(* Logix 5000 project; controller NSH_PLC1 vendor 1 type 14 code 167 rev 32.11; software revision 32.02; part 9 of 12 *)
(* tags used below, declared in another part *)
   DummyOutput : BOOL;
   LS101 : BOOL;   // Dummy Limit Switch
   MainBin1 : MainBins;   // PreClean to Huller, Main Bin #1
   MainBin2 : MainBins;   // PreClean to Huller, Main Bin #1
   MainBin3 : MainBins;   // PreClean to Huller, Main Bin #1
   MainBin4 : MainBins;   // PreClean to Huller, Main Bin #1
   MainBin5 : MainBins;   // PreClean to Huller, Main Bin #1
   MainBin6 : MainBins;   // PreClean to Huller, Main Bin #1
   MainBin7 : MainBins;   // PreClean to Huller, Main Bin #1
   MainBin8 : MainBins;   // PreClean to Huller, Main Bin #1
(* MainProgram, continued *)

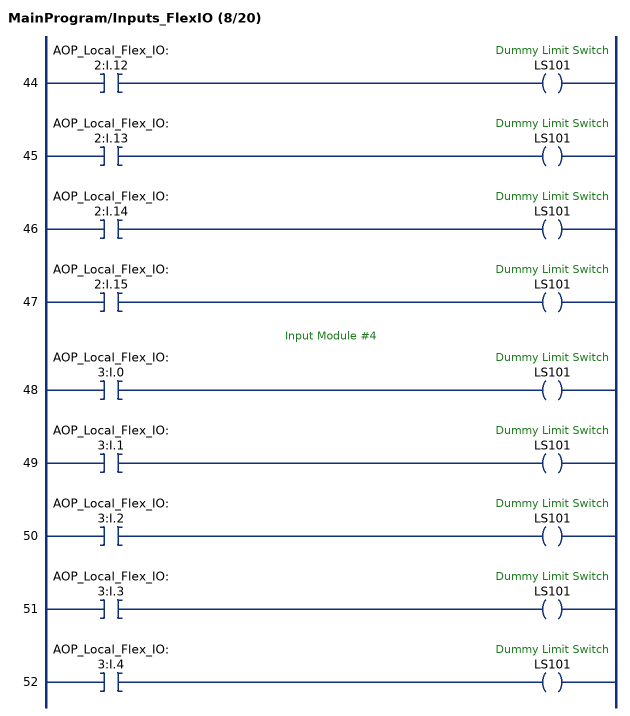
   44: XIC(AOP_Local_Flex_IO:2:I.12)OTE(LS101);
   45: XIC(AOP_Local_Flex_IO:2:I.13)OTE(LS101);
   46: XIC(AOP_Local_Flex_IO:2:I.14)OTE(LS101);
   47: XIC(AOP_Local_Flex_IO:2:I.15)OTE(LS101);
   // Input Module #4
   48: XIC(AOP_Local_Flex_IO:3:I.0)OTE(LS101);
   49: XIC(AOP_Local_Flex_IO:3:I.1)OTE(LS101);
   50: XIC(AOP_Local_Flex_IO:3:I.2)OTE(LS101);
   51: XIC(AOP_Local_Flex_IO:3:I.3)OTE(LS101);
   52: XIC(AOP_Local_Flex_IO:3:I.4)OTE(LS101);
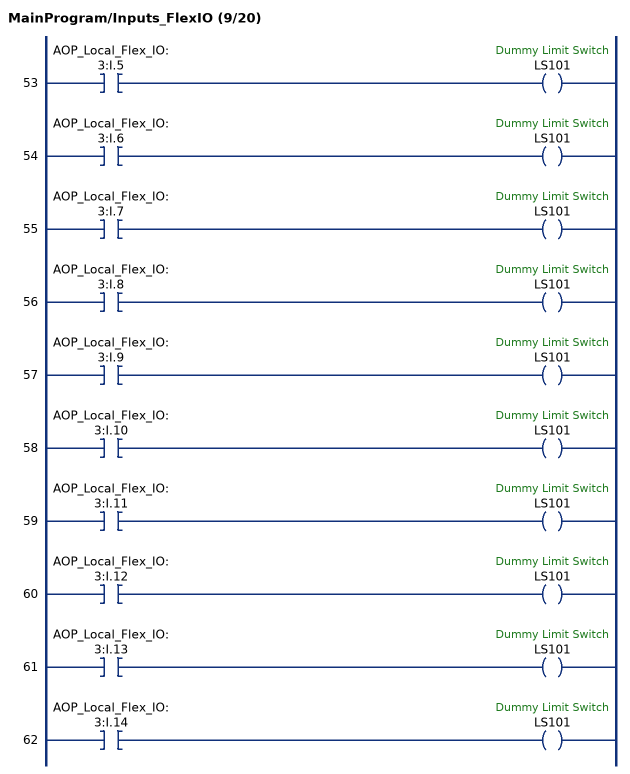
   53: XIC(AOP_Local_Flex_IO:3:I.5)OTE(LS101);
   54: XIC(AOP_Local_Flex_IO:3:I.6)OTE(LS101);
   55: XIC(AOP_Local_Flex_IO:3:I.7)OTE(LS101);
   56: XIC(AOP_Local_Flex_IO:3:I.8)OTE(LS101);
   57: XIC(AOP_Local_Flex_IO:3:I.9)OTE(LS101);
   58: XIC(AOP_Local_Flex_IO:3:I.10)OTE(LS101);
   59: XIC(AOP_Local_Flex_IO:3:I.11)OTE(LS101);
   60: XIC(AOP_Local_Flex_IO:3:I.12)OTE(LS101);
   61: XIC(AOP_Local_Flex_IO:3:I.13)OTE(LS101);
   62: XIC(AOP_Local_Flex_IO:3:I.14)OTE(LS101);
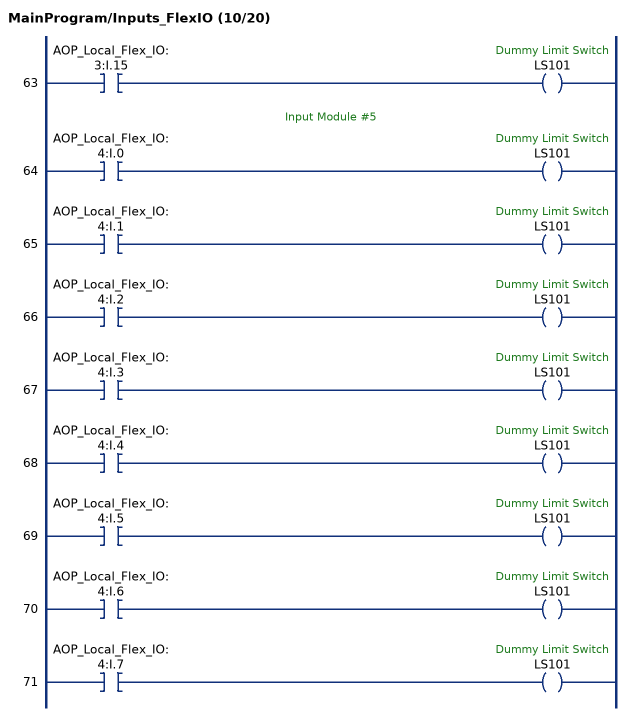
   63: XIC(AOP_Local_Flex_IO:3:I.15)OTE(LS101);
   // Input Module #5
   64: XIC(AOP_Local_Flex_IO:4:I.0)OTE(LS101);
   65: XIC(AOP_Local_Flex_IO:4:I.1)OTE(LS101);
   66: XIC(AOP_Local_Flex_IO:4:I.2)OTE(LS101);
   67: XIC(AOP_Local_Flex_IO:4:I.3)OTE(LS101);
   68: XIC(AOP_Local_Flex_IO:4:I.4)OTE(LS101);
   69: XIC(AOP_Local_Flex_IO:4:I.5)OTE(LS101);
   70: XIC(AOP_Local_Flex_IO:4:I.6)OTE(LS101);
   71: XIC(AOP_Local_Flex_IO:4:I.7)OTE(LS101);
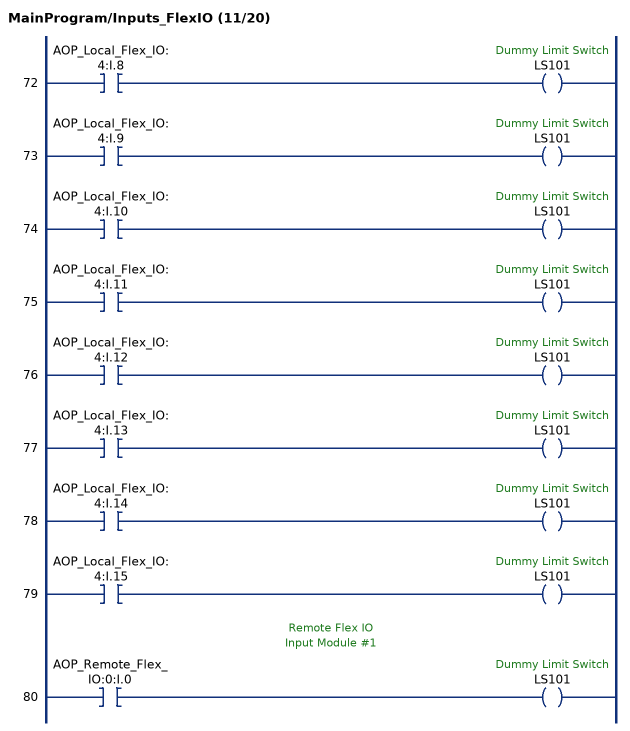
   72: XIC(AOP_Local_Flex_IO:4:I.8)OTE(LS101);
   73: XIC(AOP_Local_Flex_IO:4:I.9)OTE(LS101);
   74: XIC(AOP_Local_Flex_IO:4:I.10)OTE(LS101);
   75: XIC(AOP_Local_Flex_IO:4:I.11)OTE(LS101);
   76: XIC(AOP_Local_Flex_IO:4:I.12)OTE(LS101);
   77: XIC(AOP_Local_Flex_IO:4:I.13)OTE(LS101);
   78: XIC(AOP_Local_Flex_IO:4:I.14)OTE(LS101);
   79: XIC(AOP_Local_Flex_IO:4:I.15)OTE(LS101);
   // Remote Flex IO
   // Input Module #1
   80: XIC(AOP_Remote_Flex_IO:0:I.0)OTE(LS101);
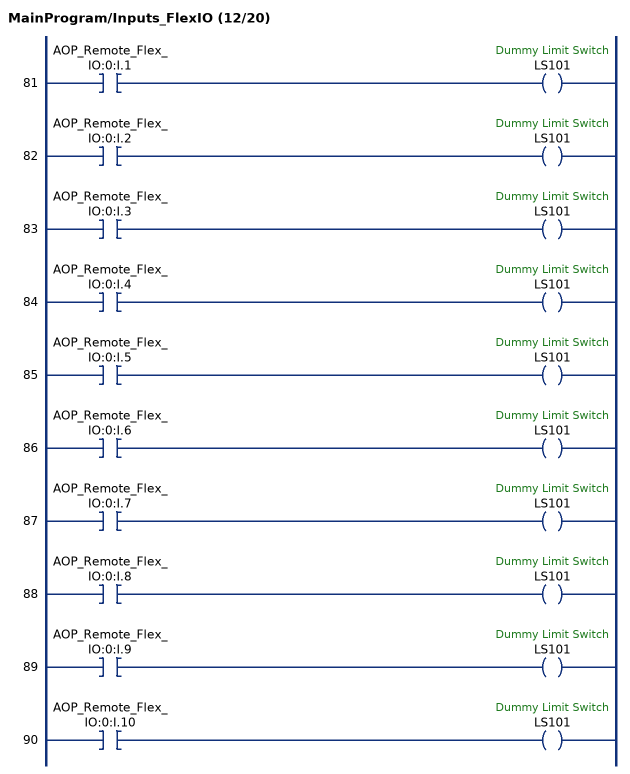
   81: XIC(AOP_Remote_Flex_IO:0:I.1)OTE(LS101);
   82: XIC(AOP_Remote_Flex_IO:0:I.2)OTE(LS101);
   83: XIC(AOP_Remote_Flex_IO:0:I.3)OTE(LS101);
   84: XIC(AOP_Remote_Flex_IO:0:I.4)OTE(LS101);
   85: XIC(AOP_Remote_Flex_IO:0:I.5)OTE(LS101);
   86: XIC(AOP_Remote_Flex_IO:0:I.6)OTE(LS101);
   87: XIC(AOP_Remote_Flex_IO:0:I.7)OTE(LS101);
   88: XIC(AOP_Remote_Flex_IO:0:I.8)OTE(LS101);
   89: XIC(AOP_Remote_Flex_IO:0:I.9)OTE(LS101);
   90: XIC(AOP_Remote_Flex_IO:0:I.10)OTE(LS101);
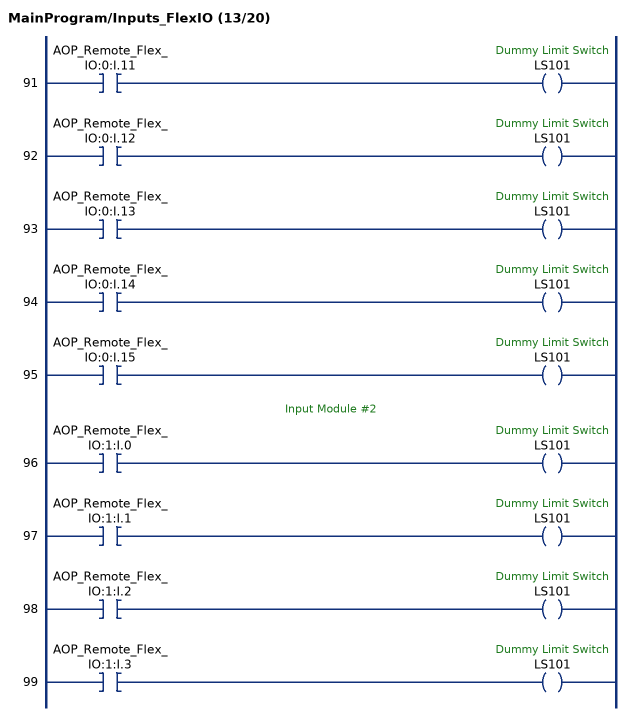
   91: XIC(AOP_Remote_Flex_IO:0:I.11)OTE(LS101);
   92: XIC(AOP_Remote_Flex_IO:0:I.12)OTE(LS101);
   93: XIC(AOP_Remote_Flex_IO:0:I.13)OTE(LS101);
   94: XIC(AOP_Remote_Flex_IO:0:I.14)OTE(LS101);
   95: XIC(AOP_Remote_Flex_IO:0:I.15)OTE(LS101);
   // Input Module #2
   96: XIC(AOP_Remote_Flex_IO:1:I.0)OTE(LS101);
   97: XIC(AOP_Remote_Flex_IO:1:I.1)OTE(LS101);
   98: XIC(AOP_Remote_Flex_IO:1:I.2)OTE(LS101);
   99: XIC(AOP_Remote_Flex_IO:1:I.3)OTE(LS101);
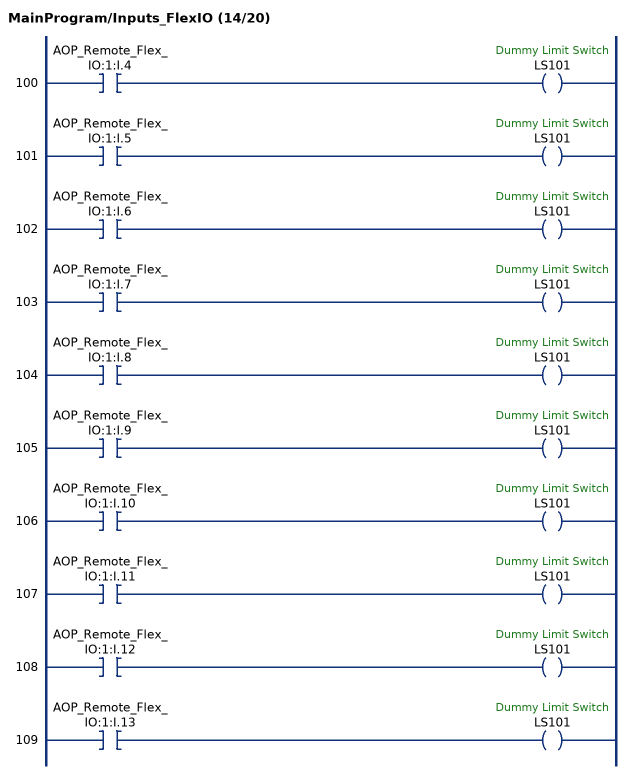
   100: XIC(AOP_Remote_Flex_IO:1:I.4)OTE(LS101);
   101: XIC(AOP_Remote_Flex_IO:1:I.5)OTE(LS101);
   102: XIC(AOP_Remote_Flex_IO:1:I.6)OTE(LS101);
   103: XIC(AOP_Remote_Flex_IO:1:I.7)OTE(LS101);
   104: XIC(AOP_Remote_Flex_IO:1:I.8)OTE(LS101);
   105: XIC(AOP_Remote_Flex_IO:1:I.9)OTE(LS101);
   106: XIC(AOP_Remote_Flex_IO:1:I.10)OTE(LS101);
   107: XIC(AOP_Remote_Flex_IO:1:I.11)OTE(LS101);
   108: XIC(AOP_Remote_Flex_IO:1:I.12)OTE(LS101);
   109: XIC(AOP_Remote_Flex_IO:1:I.13)OTE(LS101);
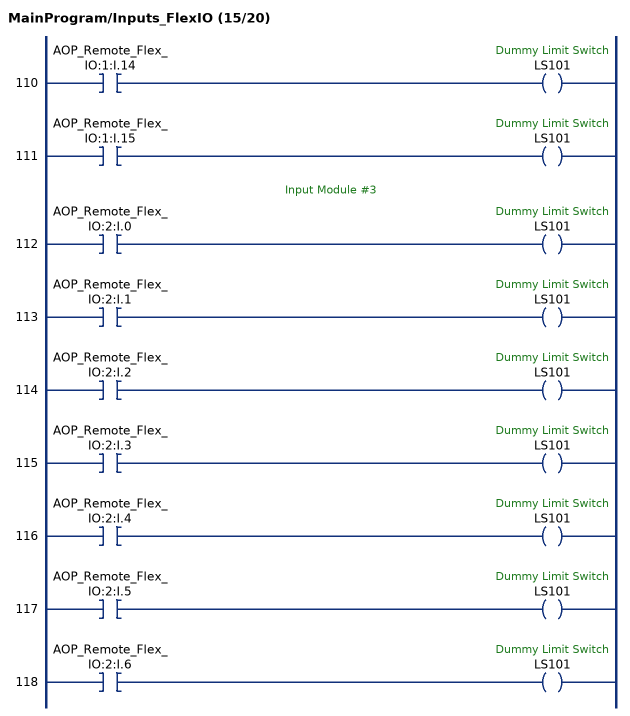
   110: XIC(AOP_Remote_Flex_IO:1:I.14)OTE(LS101);
   111: XIC(AOP_Remote_Flex_IO:1:I.15)OTE(LS101);
   // Input Module #3
   112: XIC(AOP_Remote_Flex_IO:2:I.0)OTE(LS101);
   113: XIC(AOP_Remote_Flex_IO:2:I.1)OTE(LS101);
   114: XIC(AOP_Remote_Flex_IO:2:I.2)OTE(LS101);
   115: XIC(AOP_Remote_Flex_IO:2:I.3)OTE(LS101);
   116: XIC(AOP_Remote_Flex_IO:2:I.4)OTE(LS101);
   117: XIC(AOP_Remote_Flex_IO:2:I.5)OTE(LS101);
   118: XIC(AOP_Remote_Flex_IO:2:I.6)OTE(LS101);
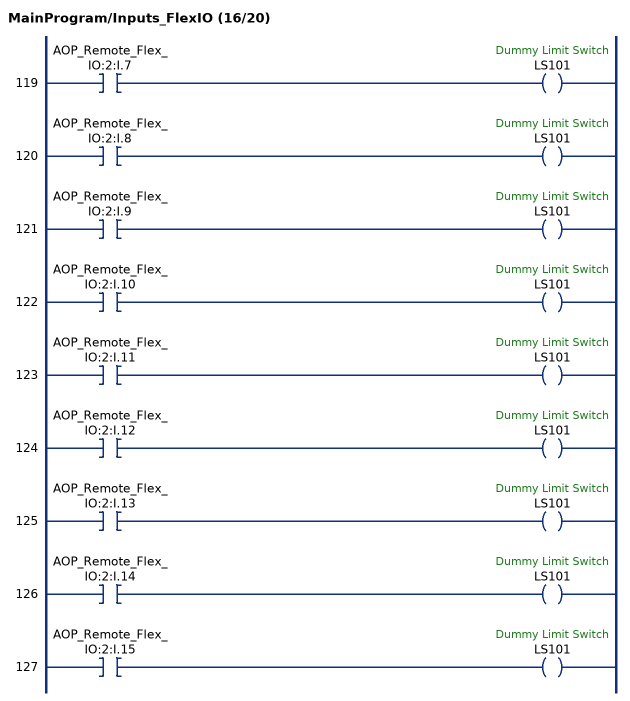
   119: XIC(AOP_Remote_Flex_IO:2:I.7)OTE(LS101);
   120: XIC(AOP_Remote_Flex_IO:2:I.8)OTE(LS101);
   121: XIC(AOP_Remote_Flex_IO:2:I.9)OTE(LS101);
   122: XIC(AOP_Remote_Flex_IO:2:I.10)OTE(LS101);
   123: XIC(AOP_Remote_Flex_IO:2:I.11)OTE(LS101);
   124: XIC(AOP_Remote_Flex_IO:2:I.12)OTE(LS101);
   125: XIC(AOP_Remote_Flex_IO:2:I.13)OTE(LS101);
   126: XIC(AOP_Remote_Flex_IO:2:I.14)OTE(LS101);
   127: XIC(AOP_Remote_Flex_IO:2:I.15)OTE(LS101);
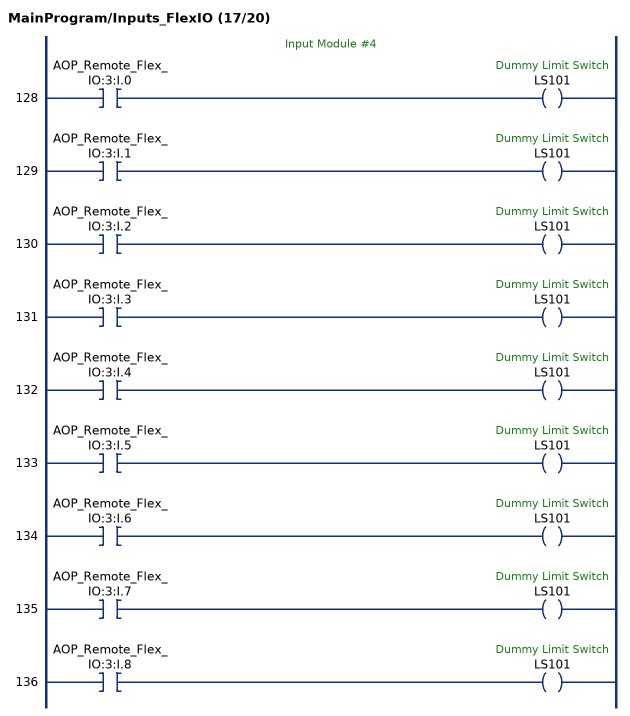
   // Input Module #4
   128: XIC(AOP_Remote_Flex_IO:3:I.0)OTE(LS101);
   129: XIC(AOP_Remote_Flex_IO:3:I.1)OTE(LS101);
   130: XIC(AOP_Remote_Flex_IO:3:I.2)OTE(LS101);
   131: XIC(AOP_Remote_Flex_IO:3:I.3)OTE(LS101);
   132: XIC(AOP_Remote_Flex_IO:3:I.4)OTE(LS101);
   133: XIC(AOP_Remote_Flex_IO:3:I.5)OTE(LS101);
   134: XIC(AOP_Remote_Flex_IO:3:I.6)OTE(LS101);
   135: XIC(AOP_Remote_Flex_IO:3:I.7)OTE(LS101);
   136: XIC(AOP_Remote_Flex_IO:3:I.8)OTE(LS101);
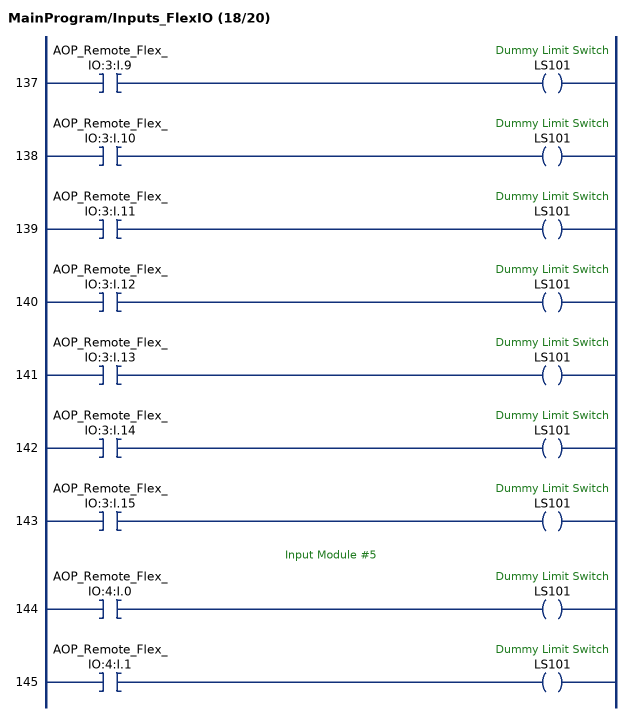
   137: XIC(AOP_Remote_Flex_IO:3:I.9)OTE(LS101);
   138: XIC(AOP_Remote_Flex_IO:3:I.10)OTE(LS101);
   139: XIC(AOP_Remote_Flex_IO:3:I.11)OTE(LS101);
   140: XIC(AOP_Remote_Flex_IO:3:I.12)OTE(LS101);
   141: XIC(AOP_Remote_Flex_IO:3:I.13)OTE(LS101);
   142: XIC(AOP_Remote_Flex_IO:3:I.14)OTE(LS101);
   143: XIC(AOP_Remote_Flex_IO:3:I.15)OTE(LS101);
   // Input Module #5
   144: XIC(AOP_Remote_Flex_IO:4:I.0)OTE(LS101);
   145: XIC(AOP_Remote_Flex_IO:4:I.1)OTE(LS101);
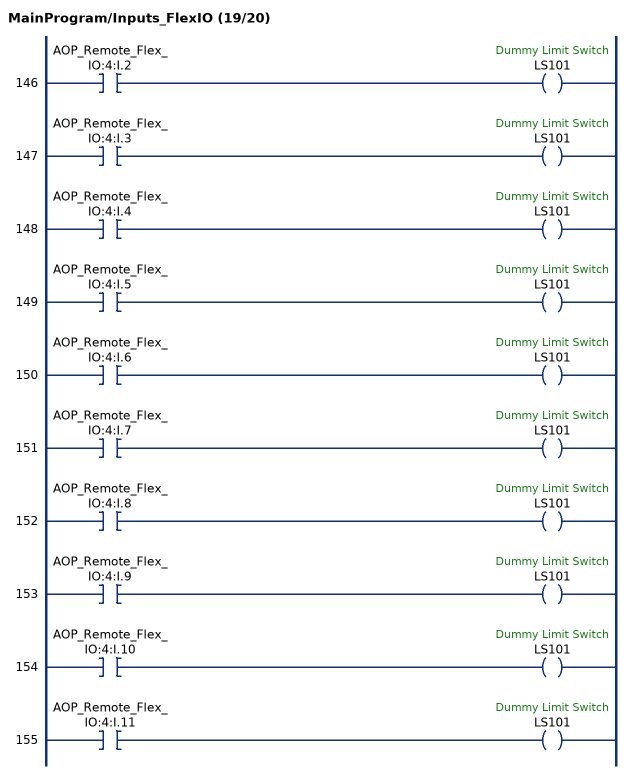
   146: XIC(AOP_Remote_Flex_IO:4:I.2)OTE(LS101);
   147: XIC(AOP_Remote_Flex_IO:4:I.3)OTE(LS101);
   148: XIC(AOP_Remote_Flex_IO:4:I.4)OTE(LS101);
   149: XIC(AOP_Remote_Flex_IO:4:I.5)OTE(LS101);
   150: XIC(AOP_Remote_Flex_IO:4:I.6)OTE(LS101);
   151: XIC(AOP_Remote_Flex_IO:4:I.7)OTE(LS101);
   152: XIC(AOP_Remote_Flex_IO:4:I.8)OTE(LS101);
   153: XIC(AOP_Remote_Flex_IO:4:I.9)OTE(LS101);
   154: XIC(AOP_Remote_Flex_IO:4:I.10)OTE(LS101);
   155: XIC(AOP_Remote_Flex_IO:4:I.11)OTE(LS101);
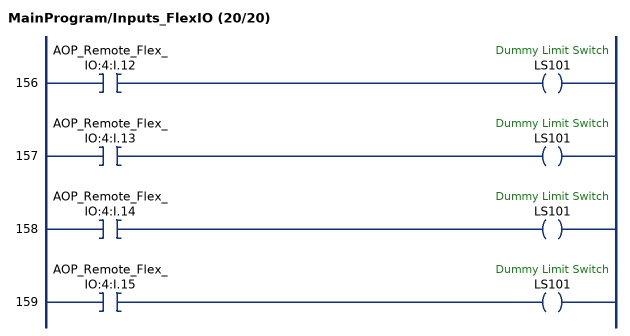
   156: XIC(AOP_Remote_Flex_IO:4:I.12)OTE(LS101);
   157: XIC(AOP_Remote_Flex_IO:4:I.13)OTE(LS101);
   158: XIC(AOP_Remote_Flex_IO:4:I.14)OTE(LS101);
   159: XIC(AOP_Remote_Flex_IO:4:I.15)OTE(LS101);
END_ROUTINE

ROUTINE Inputs_MCC1   (* ladder *)
END_ROUTINE

ROUTINE Inputs_PLC2_MCC2   (* ladder *)
END_ROUTINE

ROUTINE Inputs_PLC2_MCC3   (* ladder *)
END_ROUTINE

ROUTINE MainJSR   (* ladder *)
// Jump to Other Routines
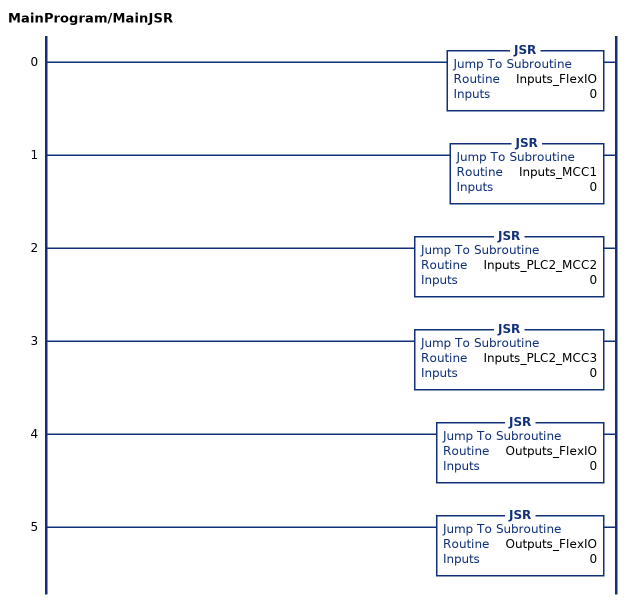
   0: JSR(Inputs_FlexIO,0);
   1: JSR(Inputs_MCC1,0);
   2: JSR(Inputs_PLC2_MCC2,0);
   3: JSR(Inputs_PLC2_MCC3,0);
   4: JSR(Outputs_FlexIO,0);
   5: JSR(Outputs_FlexIO,0);
END_ROUTINE

ROUTINE Outputs_FlexIO   (* ladder *)
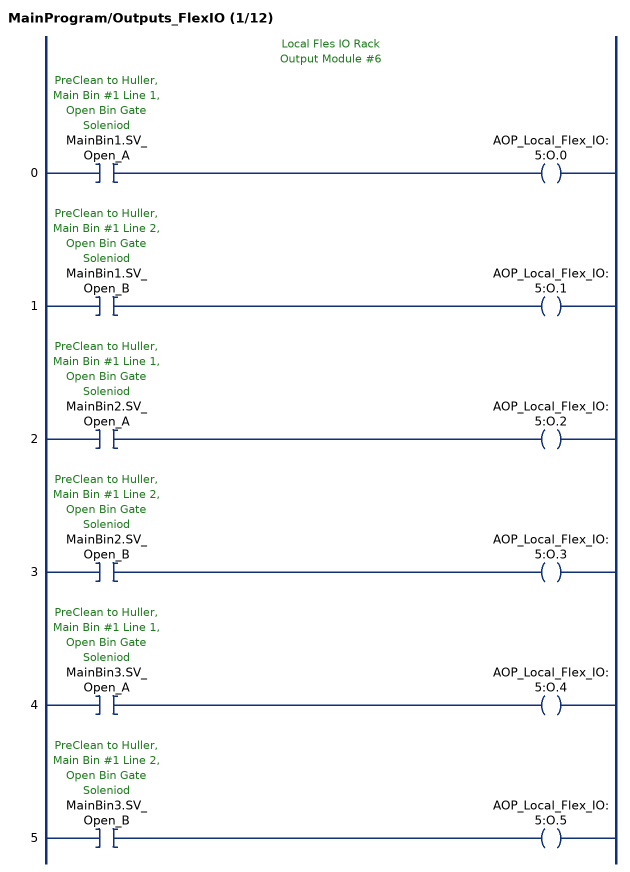
   // Local Fles IO Rack
   // Output Module #6
   0: XIC(MainBin1.SV_Open_A)OTE(AOP_Local_Flex_IO:5:O.0);
   1: XIC(MainBin1.SV_Open_B)OTE(AOP_Local_Flex_IO:5:O.1);
   2: XIC(MainBin2.SV_Open_A)OTE(AOP_Local_Flex_IO:5:O.2);
   3: XIC(MainBin2.SV_Open_B)OTE(AOP_Local_Flex_IO:5:O.3);
   4: XIC(MainBin3.SV_Open_A)OTE(AOP_Local_Flex_IO:5:O.4);
   5: XIC(MainBin3.SV_Open_B)OTE(AOP_Local_Flex_IO:5:O.5);
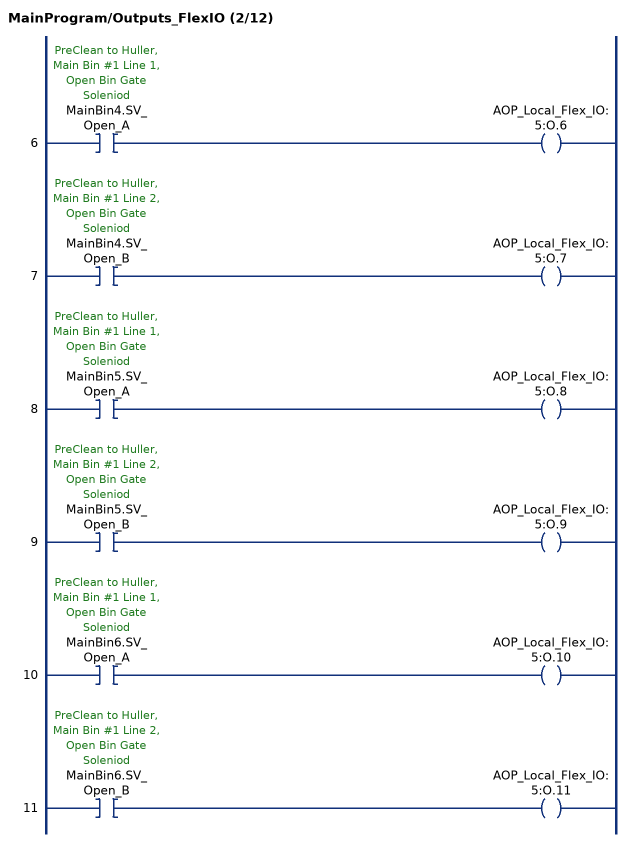
   6: XIC(MainBin4.SV_Open_A)OTE(AOP_Local_Flex_IO:5:O.6);
   7: XIC(MainBin4.SV_Open_B)OTE(AOP_Local_Flex_IO:5:O.7);
   8: XIC(MainBin5.SV_Open_A)OTE(AOP_Local_Flex_IO:5:O.8);
   9: XIC(MainBin5.SV_Open_B)OTE(AOP_Local_Flex_IO:5:O.9);
   10: XIC(MainBin6.SV_Open_A)OTE(AOP_Local_Flex_IO:5:O.10);
   11: XIC(MainBin6.SV_Open_B)OTE(AOP_Local_Flex_IO:5:O.11);
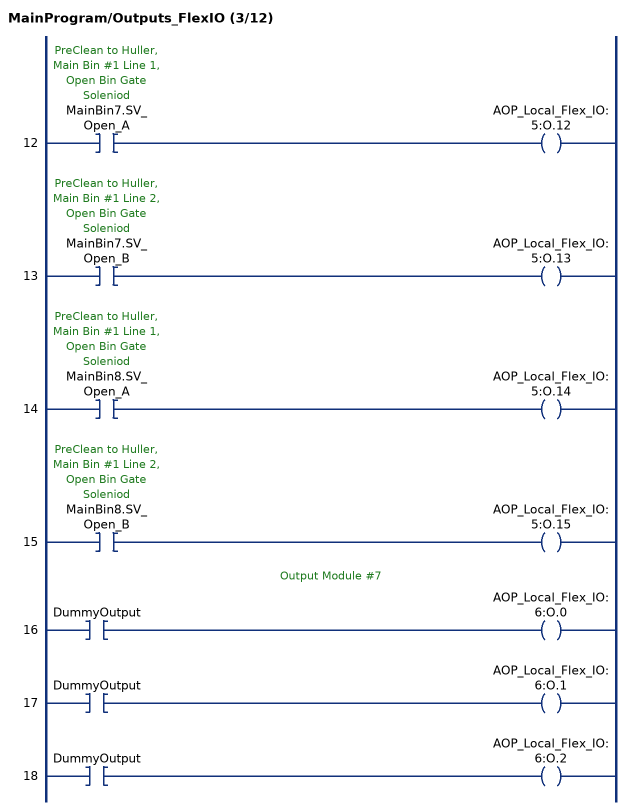
   12: XIC(MainBin7.SV_Open_A)OTE(AOP_Local_Flex_IO:5:O.12);
   13: XIC(MainBin7.SV_Open_B)OTE(AOP_Local_Flex_IO:5:O.13);
   14: XIC(MainBin8.SV_Open_A)OTE(AOP_Local_Flex_IO:5:O.14);
   15: XIC(MainBin8.SV_Open_B)OTE(AOP_Local_Flex_IO:5:O.15);
   // Output Module #7
   16: XIC(DummyOutput)OTE(AOP_Local_Flex_IO:6:O.0);
   17: XIC(DummyOutput)OTE(AOP_Local_Flex_IO:6:O.1);
   18: XIC(DummyOutput)OTE(AOP_Local_Flex_IO:6:O.2);
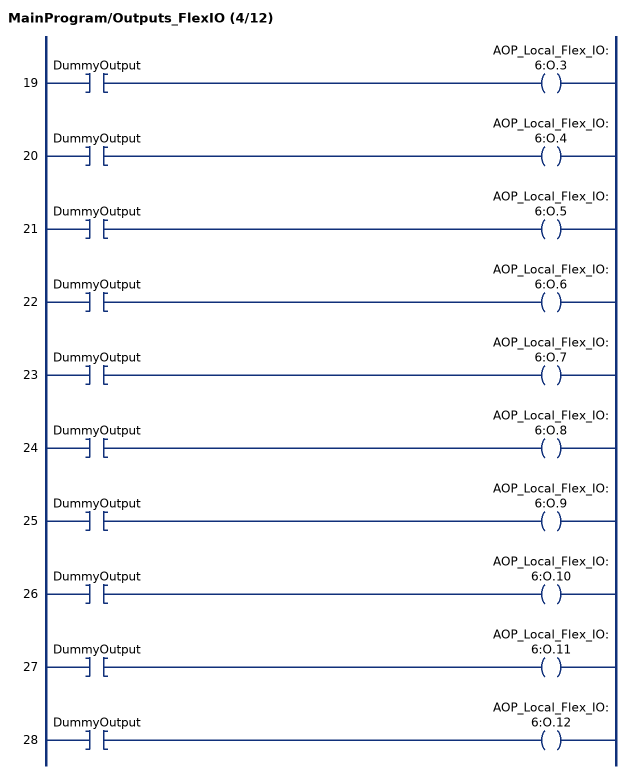
   19: XIC(DummyOutput)OTE(AOP_Local_Flex_IO:6:O.3);
   20: XIC(DummyOutput)OTE(AOP_Local_Flex_IO:6:O.4);
   21: XIC(DummyOutput)OTE(AOP_Local_Flex_IO:6:O.5);
   22: XIC(DummyOutput)OTE(AOP_Local_Flex_IO:6:O.6);
   23: XIC(DummyOutput)OTE(AOP_Local_Flex_IO:6:O.7);
   24: XIC(DummyOutput)OTE(AOP_Local_Flex_IO:6:O.8);
   25: XIC(DummyOutput)OTE(AOP_Local_Flex_IO:6:O.9);
   26: XIC(DummyOutput)OTE(AOP_Local_Flex_IO:6:O.10);
   27: XIC(DummyOutput)OTE(AOP_Local_Flex_IO:6:O.11);
   28: XIC(DummyOutput)OTE(AOP_Local_Flex_IO:6:O.12);
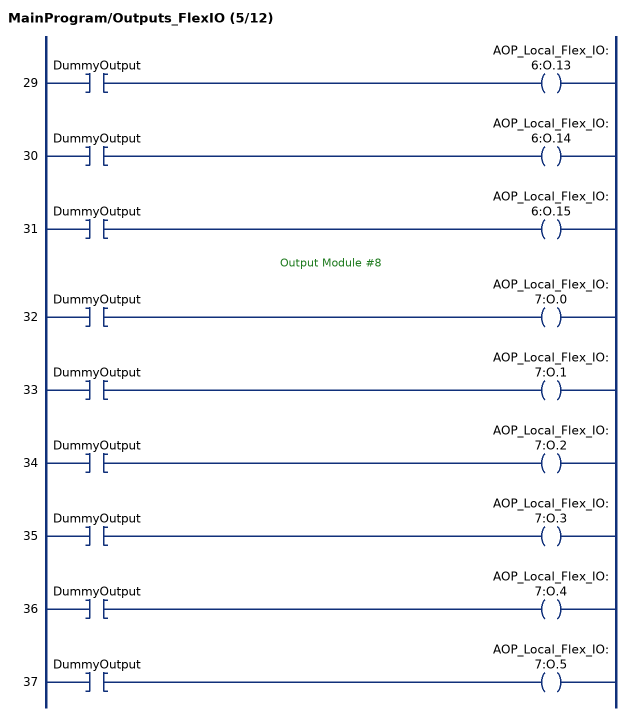
   29: XIC(DummyOutput)OTE(AOP_Local_Flex_IO:6:O.13);
   30: XIC(DummyOutput)OTE(AOP_Local_Flex_IO:6:O.14);
   31: XIC(DummyOutput)OTE(AOP_Local_Flex_IO:6:O.15);
   // Output Module #8
   32: XIC(DummyOutput)OTE(AOP_Local_Flex_IO:7:O.0);
   33: XIC(DummyOutput)OTE(AOP_Local_Flex_IO:7:O.1);
   34: XIC(DummyOutput)OTE(AOP_Local_Flex_IO:7:O.2);
   35: XIC(DummyOutput)OTE(AOP_Local_Flex_IO:7:O.3);
   36: XIC(DummyOutput)OTE(AOP_Local_Flex_IO:7:O.4);
   37: XIC(DummyOutput)OTE(AOP_Local_Flex_IO:7:O.5);
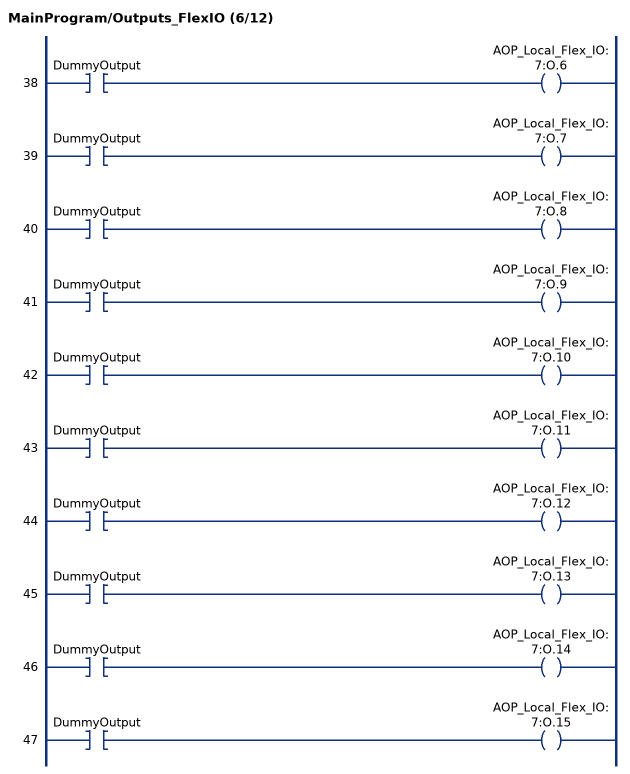
   38: XIC(DummyOutput)OTE(AOP_Local_Flex_IO:7:O.6);
   39: XIC(DummyOutput)OTE(AOP_Local_Flex_IO:7:O.7);
   40: XIC(DummyOutput)OTE(AOP_Local_Flex_IO:7:O.8);
   41: XIC(DummyOutput)OTE(AOP_Local_Flex_IO:7:O.9);
   42: XIC(DummyOutput)OTE(AOP_Local_Flex_IO:7:O.10);
   43: XIC(DummyOutput)OTE(AOP_Local_Flex_IO:7:O.11);
   44: XIC(DummyOutput)OTE(AOP_Local_Flex_IO:7:O.12);
   45: XIC(DummyOutput)OTE(AOP_Local_Flex_IO:7:O.13);
   46: XIC(DummyOutput)OTE(AOP_Local_Flex_IO:7:O.14);
   47: XIC(DummyOutput)OTE(AOP_Local_Flex_IO:7:O.15);
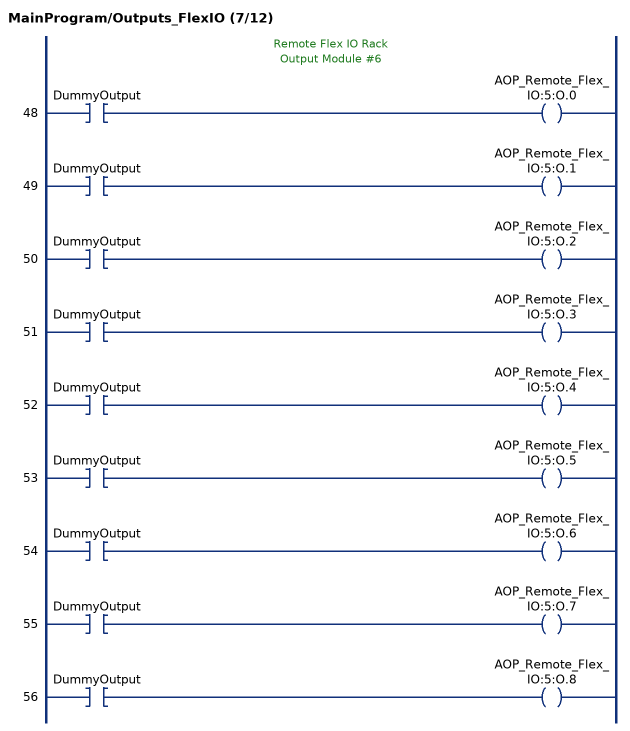
   // Remote Flex IO Rack
   // Output Module #6
   48: XIC(DummyOutput)OTE(AOP_Remote_Flex_IO:5:O.0);
   49: XIC(DummyOutput)OTE(AOP_Remote_Flex_IO:5:O.1);
   50: XIC(DummyOutput)OTE(AOP_Remote_Flex_IO:5:O.2);
   51: XIC(DummyOutput)OTE(AOP_Remote_Flex_IO:5:O.3);
   52: XIC(DummyOutput)OTE(AOP_Remote_Flex_IO:5:O.4);
   53: XIC(DummyOutput)OTE(AOP_Remote_Flex_IO:5:O.5);
   54: XIC(DummyOutput)OTE(AOP_Remote_Flex_IO:5:O.6);
   55: XIC(DummyOutput)OTE(AOP_Remote_Flex_IO:5:O.7);
   56: XIC(DummyOutput)OTE(AOP_Remote_Flex_IO:5:O.8);
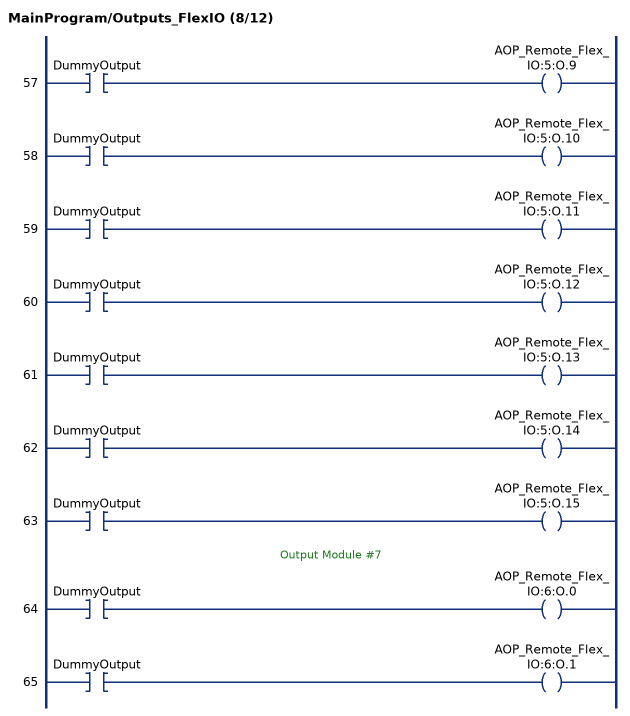
   57: XIC(DummyOutput)OTE(AOP_Remote_Flex_IO:5:O.9);
   58: XIC(DummyOutput)OTE(AOP_Remote_Flex_IO:5:O.10);
   59: XIC(DummyOutput)OTE(AOP_Remote_Flex_IO:5:O.11);
   60: XIC(DummyOutput)OTE(AOP_Remote_Flex_IO:5:O.12);
   61: XIC(DummyOutput)OTE(AOP_Remote_Flex_IO:5:O.13);
   62: XIC(DummyOutput)OTE(AOP_Remote_Flex_IO:5:O.14);
   63: XIC(DummyOutput)OTE(AOP_Remote_Flex_IO:5:O.15);
   // Output Module #7
   64: XIC(DummyOutput)OTE(AOP_Remote_Flex_IO:6:O.0);
   65: XIC(DummyOutput)OTE(AOP_Remote_Flex_IO:6:O.1);
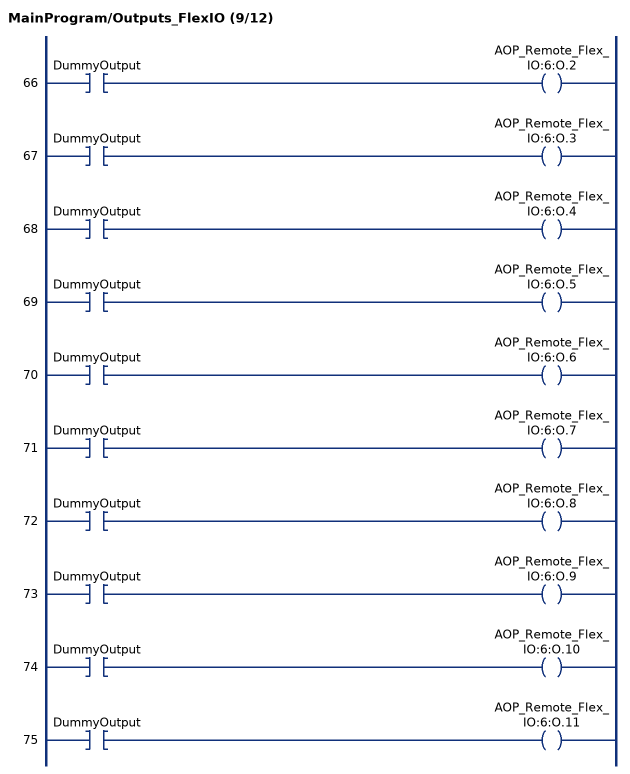
   66: XIC(DummyOutput)OTE(AOP_Remote_Flex_IO:6:O.2);
   67: XIC(DummyOutput)OTE(AOP_Remote_Flex_IO:6:O.3);
   68: XIC(DummyOutput)OTE(AOP_Remote_Flex_IO:6:O.4);
   69: XIC(DummyOutput)OTE(AOP_Remote_Flex_IO:6:O.5);
   70: XIC(DummyOutput)OTE(AOP_Remote_Flex_IO:6:O.6);
   71: XIC(DummyOutput)OTE(AOP_Remote_Flex_IO:6:O.7);
   72: XIC(DummyOutput)OTE(AOP_Remote_Flex_IO:6:O.8);
   73: XIC(DummyOutput)OTE(AOP_Remote_Flex_IO:6:O.9);
   74: XIC(DummyOutput)OTE(AOP_Remote_Flex_IO:6:O.10);
   75: XIC(DummyOutput)OTE(AOP_Remote_Flex_IO:6:O.11);
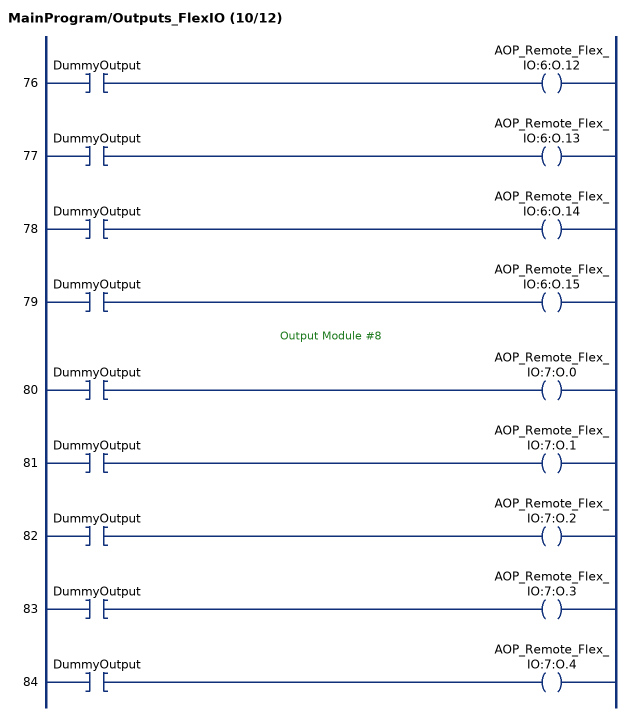
   76: XIC(DummyOutput)OTE(AOP_Remote_Flex_IO:6:O.12);
   77: XIC(DummyOutput)OTE(AOP_Remote_Flex_IO:6:O.13);
   78: XIC(DummyOutput)OTE(AOP_Remote_Flex_IO:6:O.14);
   79: XIC(DummyOutput)OTE(AOP_Remote_Flex_IO:6:O.15);
   // Output Module #8
   80: XIC(DummyOutput)OTE(AOP_Remote_Flex_IO:7:O.0);
   81: XIC(DummyOutput)OTE(AOP_Remote_Flex_IO:7:O.1);
   82: XIC(DummyOutput)OTE(AOP_Remote_Flex_IO:7:O.2);
   83: XIC(DummyOutput)OTE(AOP_Remote_Flex_IO:7:O.3);
   84: XIC(DummyOutput)OTE(AOP_Remote_Flex_IO:7:O.4);
